FUNCTION IO_CouplingAsFunction : BOOL

// will be used for IO coupling test

END_FUNCTION

(* stored: Version 1.1.0.1, ProductVersion 3.1.4024.12
   POU IO_CouplingAsFunction: Id {51cf6aa0-f974-4546-be43-88ca6f6efa73}, SpecialFunc None *)
